FUNCTION_BLOCK RunInputV1 EXTENDS RunUnitSlave
VAR_INPUT
	handy : BOOL; //link to handy(on)
	lightScreen : BOOL; //link to light screen
		
	materialRemains : UINT; //link to the counter of all controllers
	
	materialValidSensor : BOOL; //link to approximity
END_VAR
VAR_OUTPUT
	inputCounter : UINT;
END_VAR
VAR
	clamper : POINTER TO RunCylinder;
	
	controller : POINTER TO RunUnitController; //link to parent
	toggleClear : BOOL; // link to HMI clear request
END_VAR

SUPER^();

//status backup
IF NOT toggleClear AND (controller<>0 AND_THEN controller^.interfaceControl^.materialClear) THEN
	toggleClear := TRUE;
END_IF

CASE outputState OF
	eSpecialStates.SLAVE_ENTER_PROCEDURE:
		bSerialTransition := clamper^.Execute(eCylinderCommands.COMMAND_B); //release
	16#201:
		//wait until trigger off
		bSerialTransition := NOT handy;
		IF bSerialTransition THEN
			SlotBase^.Valid := FALSE; //reset
		END_IF
		//
		IF toggleClear AND materialRemains = 0 THEN
			toggleClear := FALSE;
		END_IF
	16#202:
		//conditions
		//1. bypassed
		//2. handy on
		//3. toggle clear
		//4. material existed with light screen off
		IF toggleClear OR bIsBypassed OR handy OR ( lightScreen AND SlotBase^.Valid) THEN
			bSerialTransition := TRUE;
		END_IF
		//once material detected , clamper imdiatly
		IF NOT SlotBase^.Valid AND materialValidSensor THEN
			clamper^.Execute(eCylinderCommands.COMMAND_A);
			SlotBase^.Valid := TRUE;
			//count-up
			inputCounter := inputCounter + 1;
			// material transfer
			SlotBase^.Act := TRUE;
		END_IF
	16#203:
		IF clamper^.Execute(eCylinderCommands.COMMAND_A) THEN
			//closure
			NextState := eSpecialStates.SLAVE_WORK_DONE;
		END_IF
END_CASE

METHOD FB_init : BOOL
VAR_INPUT
	bInitRetains : BOOL; // if TRUE, the retain variables are initialized (warm start / cold start)
	bInCopyCode : BOOL;  // if TRUE, the instance afterwards gets moved into the copy code (online change)
	
	argParent : POINTER TO RunUnitGeneric;
	argSlotBase : POINTER TO RunMaterial;
	argSlotLast : POINTER TO RunMaterial;
	
	argWorkingSignal : POINTER TO BOOL;
	
	argClamper : POINTER TO RunCylinder;
END_VAR
//initialize 
Parent := argParent;
SlotBase := argSlotBase;
SlotLast := argSlotLast;
//
IF bInitRetains THEN
	NextState := eSpecialStates.INITIAL_BEGIN;
END_IF

controller := Parent;

workingSignal := argWorkingSignal; //link
//link
clamper := argClamper;
END_METHOD

METHOD Initialize : BOOL
VAR_INPUT
END_VAR

CASE outputState OF
	eSpecialStates.INITIAL_BEGIN:
		IF clamper^.Execute(eCylinderCommands.COMMAND_A) THEN
			//release clamper
			NextState := eSpecialStates.INITIAL_END;
		END_IF
END_CASE

Initialize := SUPER^.Initialize();
END_METHOD

END_FUNCTION_BLOCK

(* stored: Version 1.1.0.1, ProductVersion 3.1.4024.0
   POU RunInputV1: Id {68b3e97e-d64b-4e62-becb-dd70186a6197}, SpecialFunc None
   Method FB_init: Id {6e9ca68a-b2aa-44f6-88fb-ae41aaca9008}
   Method Initialize: Id {71942685-e4a4-4702-ac08-2d35b3a9e76b} *)
